// SIMATIC S7-200 SMART project (STEP 7-Micro/WIN SMART), CPU ST40

SYMBOL_TABLE 用户定义1
D1GD             I0.0     // 道1光电
D2GD             I0.1     // 道2光电
D3GD             I0.2     // 道3光电
D4GD             I0.3     // 道4光电
D1YX             I0.4     // 道1运行
D2YX             I0.5     // 道2运行
D3YX             I0.6     // 道3运行
D4YX             I0.7     // 道4运行
END_SYMBOL_TABLE

SYMBOL_TABLE 系统符号
Always_On        SM0.0    // 始终接通
First_Scan_On    SM0.1    // 仅在第一个扫描周期时接通
Clock_1s         SM0.5    // 针对 1 s 的周期时间，时钟脉冲接通 0.5 s，断开 0.5 s.
P0_Config        SMB30    // 组态端口 0 通信：奇偶校验、每个字符的数据位数、波特率和协议
END_SYMBOL_TABLE

SYMBOL_TABLE TCPServer1
State            VB5000
SendBuffer       VB5100
RecvBuffer       VB5300
RecvLenth        VW5004
SendLenth        VW5006
SendBufferW      VW5100
RecvBufferW      VW5300
StateConnect     1
StateConnectWait 2
StateTransmit    3
StateTransmitWait 4
StateReceive     5
StateRecvCheck   6
StateDisconnect  7
StateDisconnectWait 8
ExitSwitch       10
SendLenthB       VB5008
END_SYMBOL_TABLE

ORGANIZATION_BLOCK 主程序:OB1
TITLE=程序注释
BEGIN
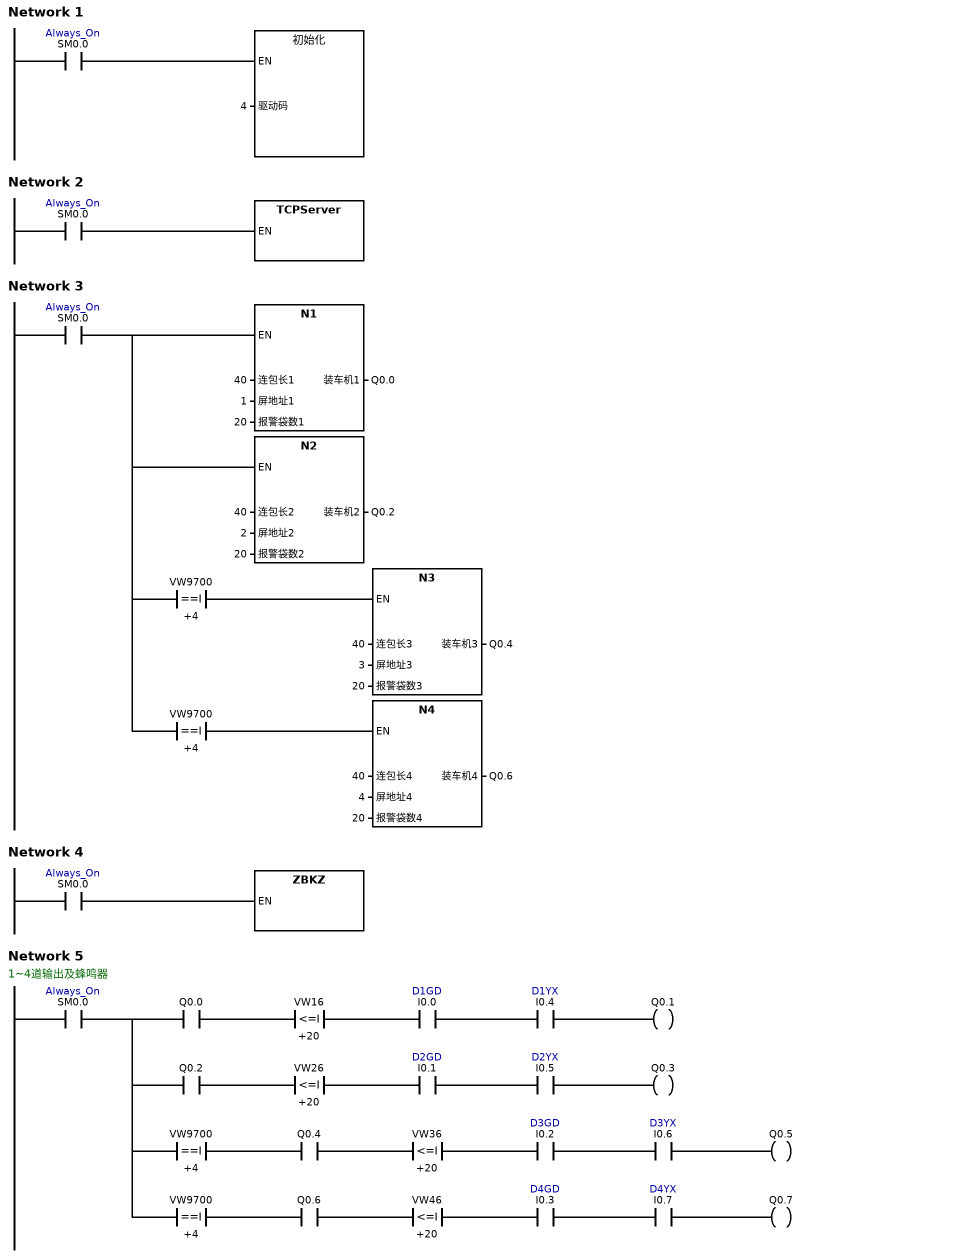
Network 1
LD     Always_On:SM0.0
CALL   初始化:SBR0, 4
Network 2
LD     Always_On:SM0.0
CALL   TCPServer:SBR50
Network 3
LD     Always_On:SM0.0
LPS
CALL   N1:SBR1, 40, 1, 20, Q0.0
CALL   N2:SBR2, 40, 2, 20, Q0.2
AW=    VW9700, +4
CALL   N3:SBR3, 40, 3, 20, Q0.4
LPP
AW=    VW9700, +4
CALL   N4:SBR4, 40, 4, 20, Q0.6
Network 4
LD     Always_On:SM0.0
CALL   ZBKZ:SBR9
Network 5
// 1~4道输出及蜂鸣器
LD     Always_On:SM0.0
LPS
A      Q0.0
AW<=   VW16, +20
A      D1GD:I0.0
A      D1YX:I0.4
=      Q0.1
LRD
A      Q0.2
AW<=   VW26, +20
A      D2GD:I0.1
A      D2YX:I0.5
=      Q0.3
LRD
AW=    VW9700, +4
A      Q0.4
AW<=   VW36, +20
A      D3GD:I0.2
A      D3YX:I0.6
=      Q0.5
LPP
AW=    VW9700, +4
A      Q0.6
AW<=   VW46, +20
A      D4GD:I0.3
A      D4YX:I0.7
=      Q0.7
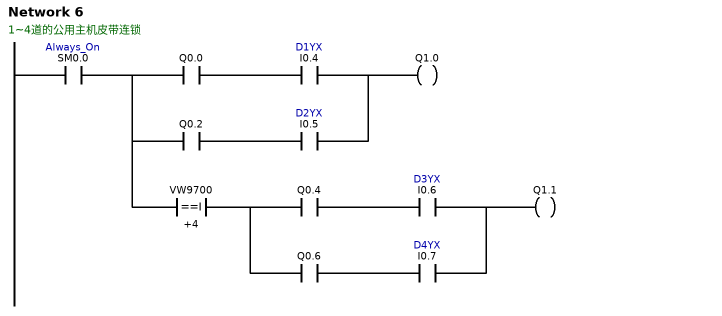
Network 6
// 1~4道的公用主机皮带连锁
LD     Always_On:SM0.0
LPS
LD     Q0.0
A      D1YX:I0.4
LD     Q0.2
A      D2YX:I0.5
OLD
ALD
=      Q1.0
LPP
AW=    VW9700, +4
LD     Q0.4
A      D3YX:I0.6
LD     Q0.6
A      D4YX:I0.7
OLD
ALD
=      Q1.1
END_ORGANIZATION_BLOCK

SUBROUTINE_BLOCK 初始化:SBR0
TITLE=子程序注释
VAR_INPUT
驱动码:WORD;	// LW0 
END_VAR
VAR
temp1:WORD;	// LW2 
temp2:WORD;	// LW4 
END_VAR
BEGIN
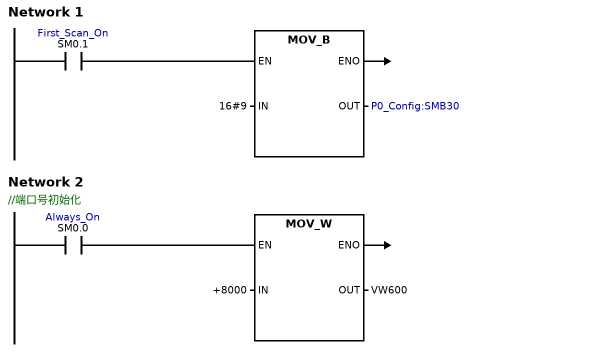
Network 1
// 首次扫描时，
// 初始化自由端口：
// - 选择9600波特
// - 选择8个数据位
// - 选择无校验
// 初始化RCV信息控制字节：
// - RCV被启用
// - 检测到信息字符结束
// - 将空闲行条件检测为
// 信息开始条件。
// 将信息字符结束设为hex OA（换行符）。
// 将空闲行超时设为5毫秒。
// 将最大字符数设为100。
// 为端口0在VB100位置启用带缓冲区的接收方框
LD     First_Scan_On:SM0.1
MOVB   16#9, P0_Config:SMB30
Network 2
// //端口号初始化
LD     Always_On:SM0.0
MOVW   +8000, VW600
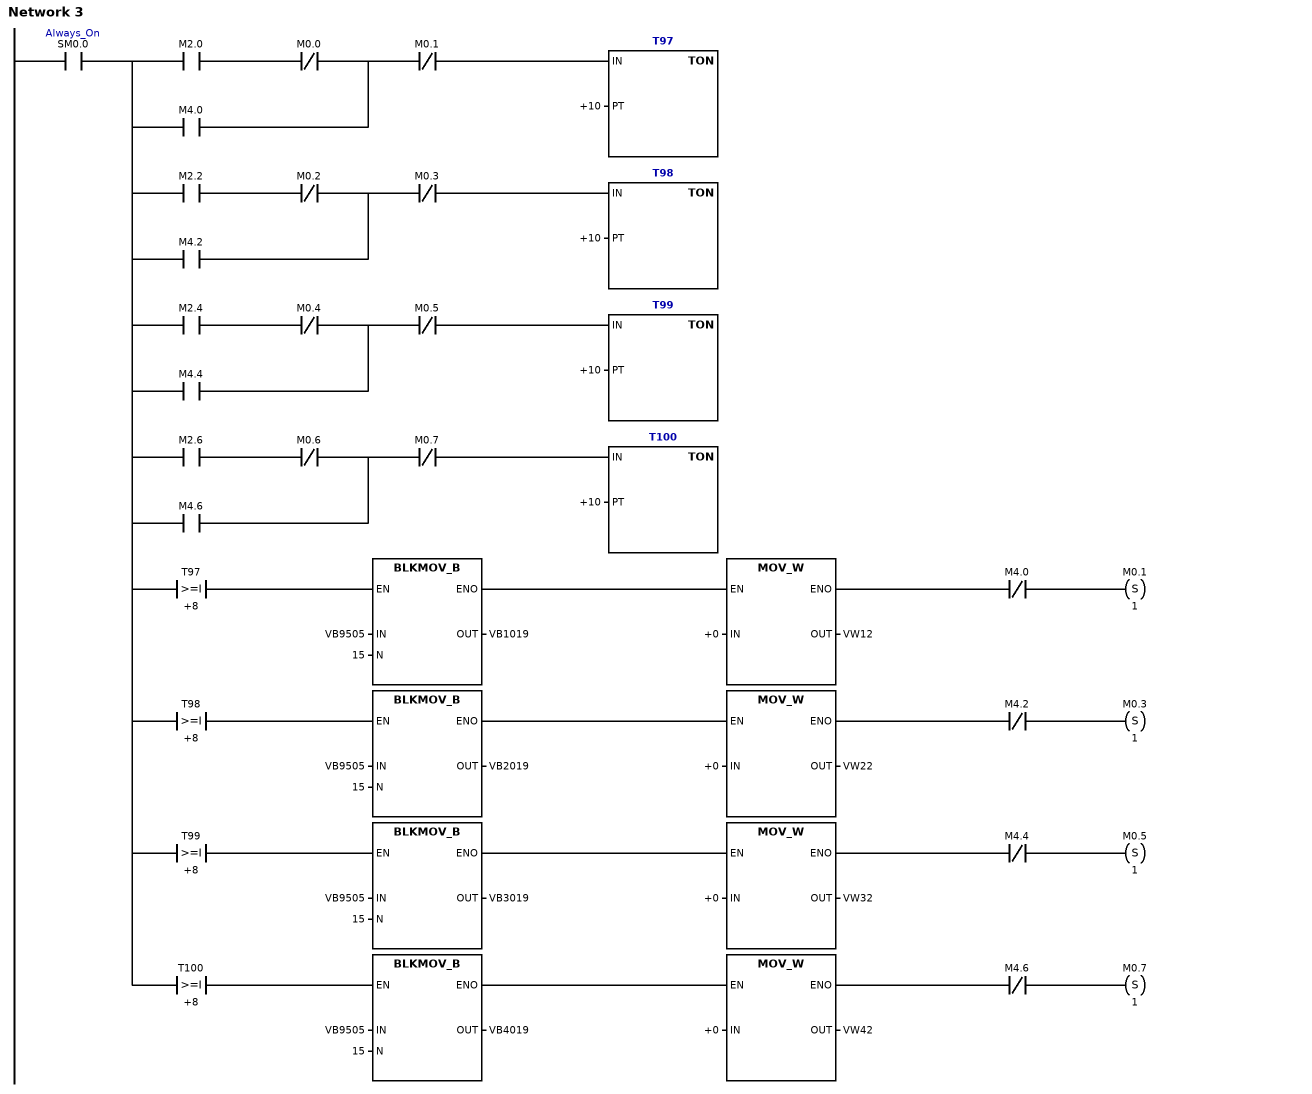
Network 3
LD     Always_On:SM0.0
LPS
LD     M2.0
AN     M0.0
O      M4.0
ALD
AN     M0.1
TON    T97, +10
LRD
LD     M2.2
AN     M0.2
O      M4.2
ALD
AN     M0.3
TON    T98, +10
LRD
LD     M2.4
AN     M0.4
O      M4.4
ALD
AN     M0.5
TON    T99, +10
LRD
LD     M2.6
AN     M0.6
O      M4.6
ALD
AN     M0.7
TON    T100, +10
LPP
LPS
AW>=   T97, +8
BMB    VB9505, VB1019, 15
AENO
MOVW   +0, VW12
AENO
AN     M4.0
S      M0.1, 1
LRD
AW>=   T98, +8
BMB    VB9505, VB2019, 15
AENO
MOVW   +0, VW22
AENO
AN     M4.2
S      M0.3, 1
LRD
AW>=   T99, +8
BMB    VB9505, VB3019, 15
AENO
MOVW   +0, VW32
AENO
AN     M4.4
S      M0.5, 1
LPP
AW>=   T100, +8
BMB    VB9505, VB4019, 15
AENO
MOVW   +0, VW42
AENO
AN     M4.6
S      M0.7, 1
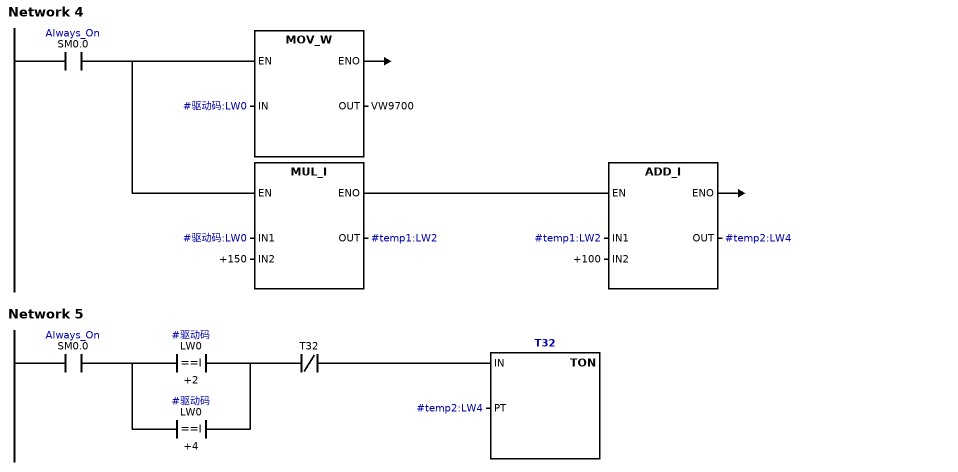
Network 4
LD     Always_On:SM0.0
MOVW   #驱动码:LW0, VW9700
MOVW   #驱动码:LW0, #temp1:LW2
AENO
*I     +150, #temp1:LW2
AENO
MOVW   #temp1:LW2, #temp2:LW4
+I     +100, #temp2:LW4
Network 5
LD     Always_On:SM0.0
LDW=   #驱动码:LW0, +2
OW=    #驱动码:LW0, +4
ALD
AN     T32
TON    T32, #temp2:LW4
END_SUBROUTINE_BLOCK

SUBROUTINE_BLOCK N1:SBR1
TITLE=
VAR_INPUT
连包长1:WORD;	// LW0 
屏地址1:BYTE;	// LB2 
报警袋数1:WORD;	// LW3 
END_VAR
VAR_OUTPUT
装车机1:BOOL;	// L5.0 
END_VAR
VAR
总袋数1:WORD;	// LW6 
袋长1:WORD;	// LW8 
已装袋数1:WORD;	// LW10 
剩余袋数1:WORD;	// LW12 
END_VAR
BEGIN
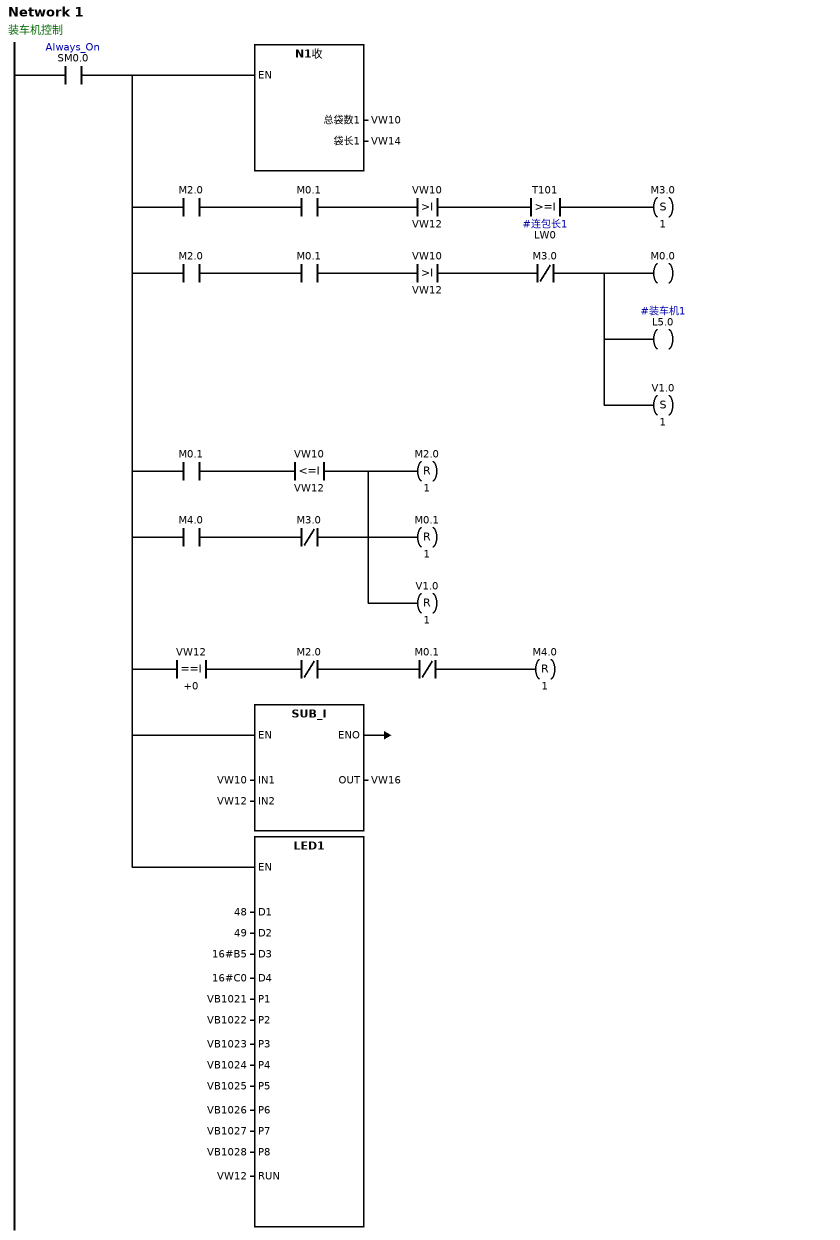
Network 1
// 装车机控制
LD     Always_On:SM0.0
LPS
CALL   N1收:SBR21, VW10, VW14
A      M2.0
A      M0.1
AW>    VW10, VW12
AW>=   T101, #连包长1:LW0
S      M3.0, 1
LRD
A      M2.0
A      M0.1
AW>    VW10, VW12
AN     M3.0
=      M0.0
=      #装车机1:L5.0
S      V1.0, 1
LRD
LD     M0.1
AW<=   VW10, VW12
LD     M4.0
AN     M3.0
OLD
ALD
R      M2.0, 1
R      M0.1, 1
R      V1.0, 1
LPP
LPS
AW=    VW12, +0
AN     M2.0
AN     M0.1
R      M4.0, 1
LRD
MOVW   VW10, VW16
-I     VW12, VW16
LPP
CALL   LED1:SBR11, 48, 49, 16#B5, 16#C0, VB1021, VB1022, VB1023, VB1024, VB1025, VB1026, VB1027, VB1028, VW12
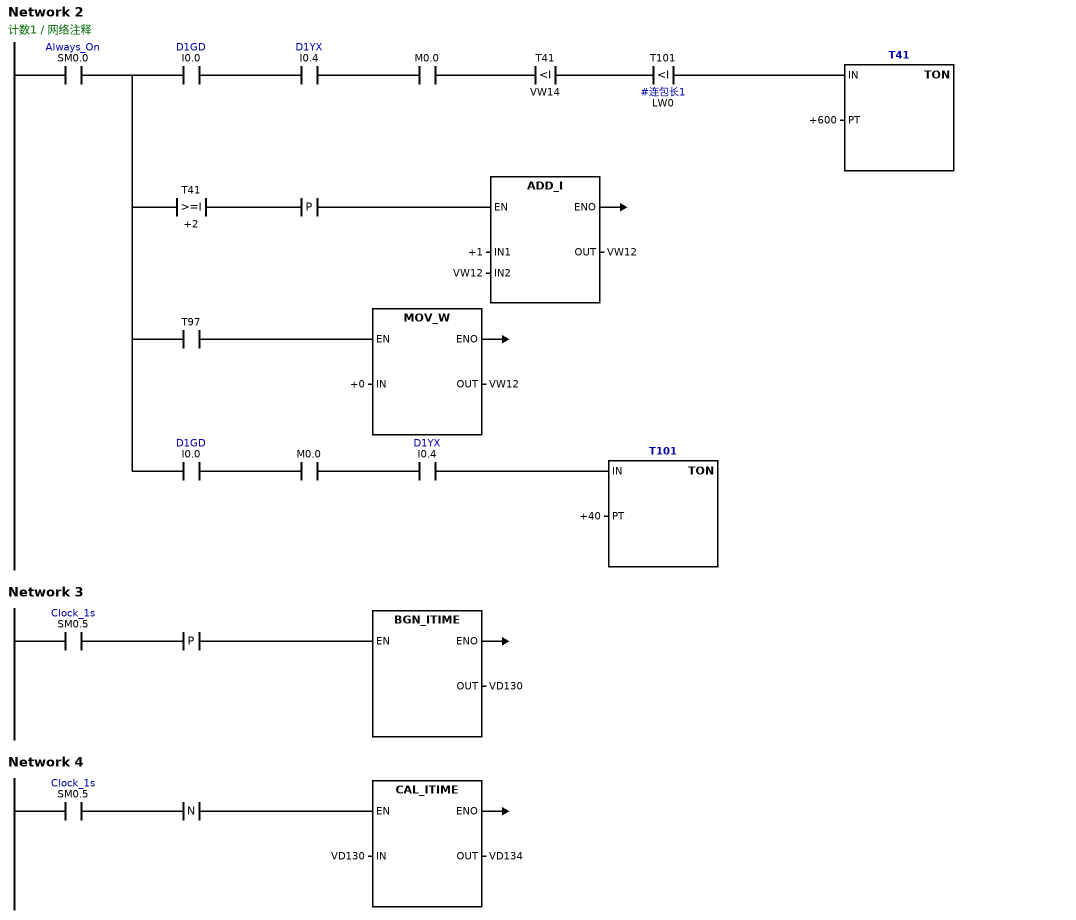
Network 2
// 计数1
// 网络注释
LD     Always_On:SM0.0
LPS
A      D1GD:I0.0
A      D1YX:I0.4
A      M0.0
AW<    T41, VW14
AW<    T101, #连包长1:LW0
TON    T41, +600
LRD
AW>=   T41, +2
EU
+I     +1, VW12
LRD
A      T97
MOVW   +0, VW12
LPP
A      D1GD:I0.0
A      M0.0
A      D1YX:I0.4
TON    T101, +40
Network 3
LD     Clock_1s:SM0.5
EU
BITIM  VD130
Network 4
LD     Clock_1s:SM0.5
ED
CITIM  VD130, VD134
END_SUBROUTINE_BLOCK

SUBROUTINE_BLOCK N2:SBR2
TITLE=
VAR_INPUT
连包长2:WORD;	// LW0 
屏地址2:BYTE;	// LB2 
报警袋数2:WORD;	// LW3 
END_VAR
VAR_OUTPUT
装车机2:BOOL;	// L5.0 
END_VAR
VAR
总袋数2:WORD;	// LW6 
袋长2:WORD;	// LW8 
已装袋数2:WORD;	// LW10 
剩余袋数2:WORD;	// LW12 
END_VAR
BEGIN
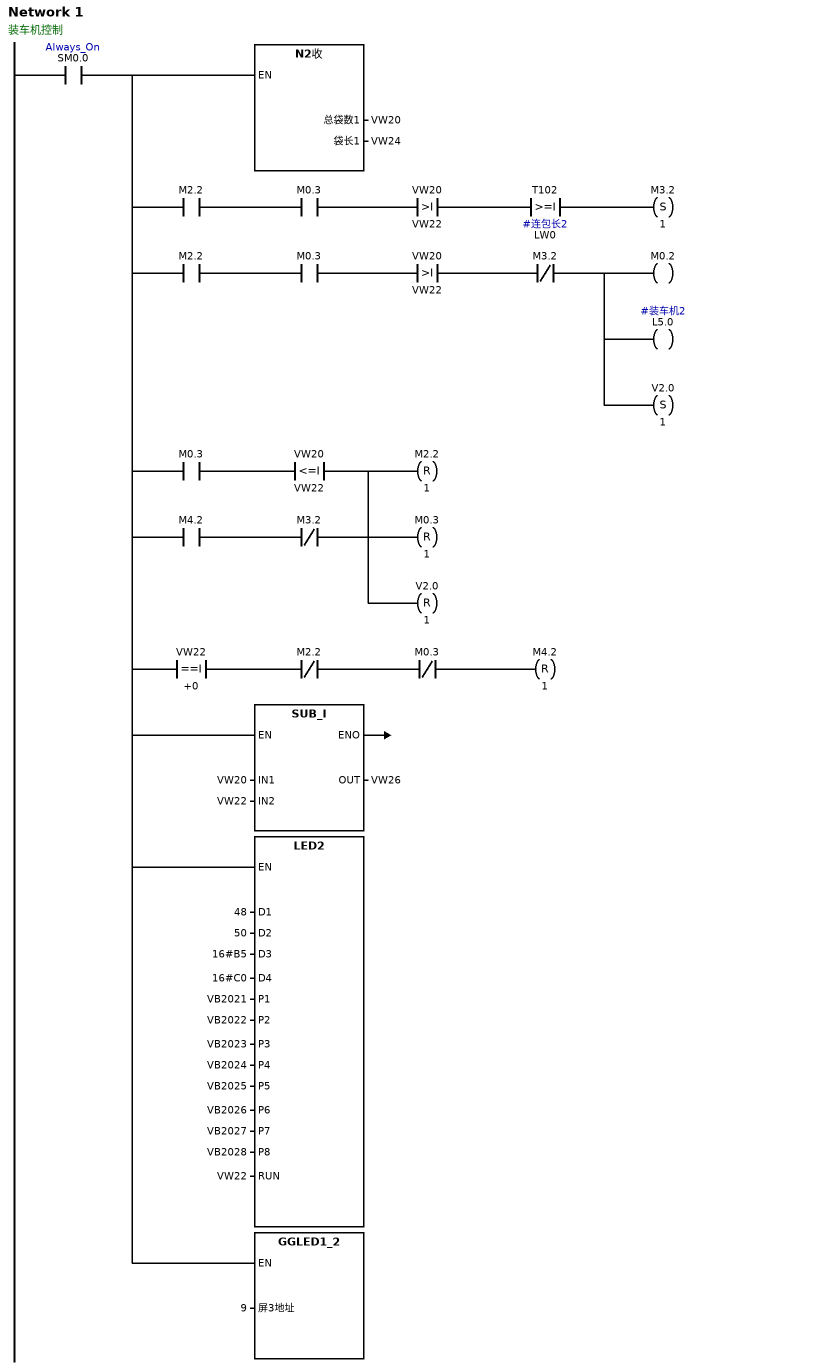
Network 1
// 装车机控制
LD     Always_On:SM0.0
LPS
CALL   N2收:SBR22, VW20, VW24
A      M2.2
A      M0.3
AW>    VW20, VW22
AW>=   T102, #连包长2:LW0
S      M3.2, 1
LRD
A      M2.2
A      M0.3
AW>    VW20, VW22
AN     M3.2
=      M0.2
=      #装车机2:L5.0
S      V2.0, 1
LRD
LD     M0.3
AW<=   VW20, VW22
LD     M4.2
AN     M3.2
OLD
ALD
R      M2.2, 1
R      M0.3, 1
R      V2.0, 1
LPP
LPS
AW=    VW22, +0
AN     M2.2
AN     M0.3
R      M4.2, 1
LRD
MOVW   VW20, VW26
-I     VW22, VW26
LRD
CALL   LED2:SBR12, 48, 50, 16#B5, 16#C0, VB2021, VB2022, VB2023, VB2024, VB2025, VB2026, VB2027, VB2028, VW22
LPP
CALL   GGLED1_2:SBR31, 9
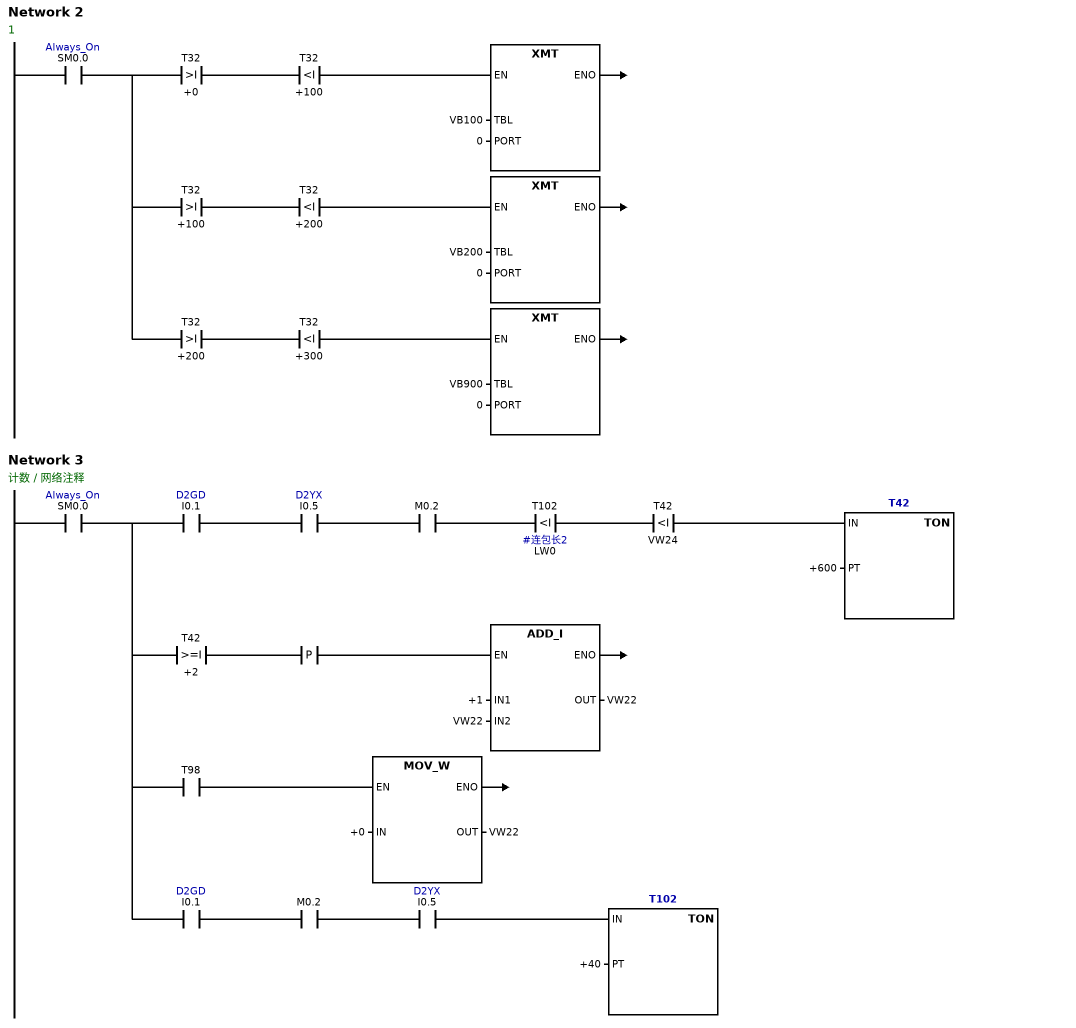
Network 2
// 1
LD     Always_On:SM0.0
LPS
AW>    T32, +0
AW<    T32, +100
XMT    VB100, 0
LRD
AW>    T32, +100
AW<    T32, +200
XMT    VB200, 0
LPP
AW>    T32, +200
AW<    T32, +300
XMT    VB900, 0
Network 3
// 计数
// 网络注释
LD     Always_On:SM0.0
LPS
A      D2GD:I0.1
A      D2YX:I0.5
A      M0.2
AW<    T102, #连包长2:LW0
AW<    T42, VW24
TON    T42, +600
LRD
AW>=   T42, +2
EU
+I     +1, VW22
LRD
A      T98
MOVW   +0, VW22
LPP
A      D2GD:I0.1
A      M0.2
A      D2YX:I0.5
TON    T102, +40
END_SUBROUTINE_BLOCK

SUBROUTINE_BLOCK N3:SBR3
TITLE=
VAR_INPUT
连包长3:WORD;	// LW0 
屏地址3:BYTE;	// LB2 
报警袋数3:WORD;	// LW3 
END_VAR
VAR_OUTPUT
装车机3:BOOL;	// L5.0 
END_VAR
VAR
总袋数3:WORD;	// LW6 
袋长3:WORD;	// LW8 
已装袋数3:WORD;	// LW10 
剩余袋数3:WORD;	// LW12 
END_VAR
BEGIN
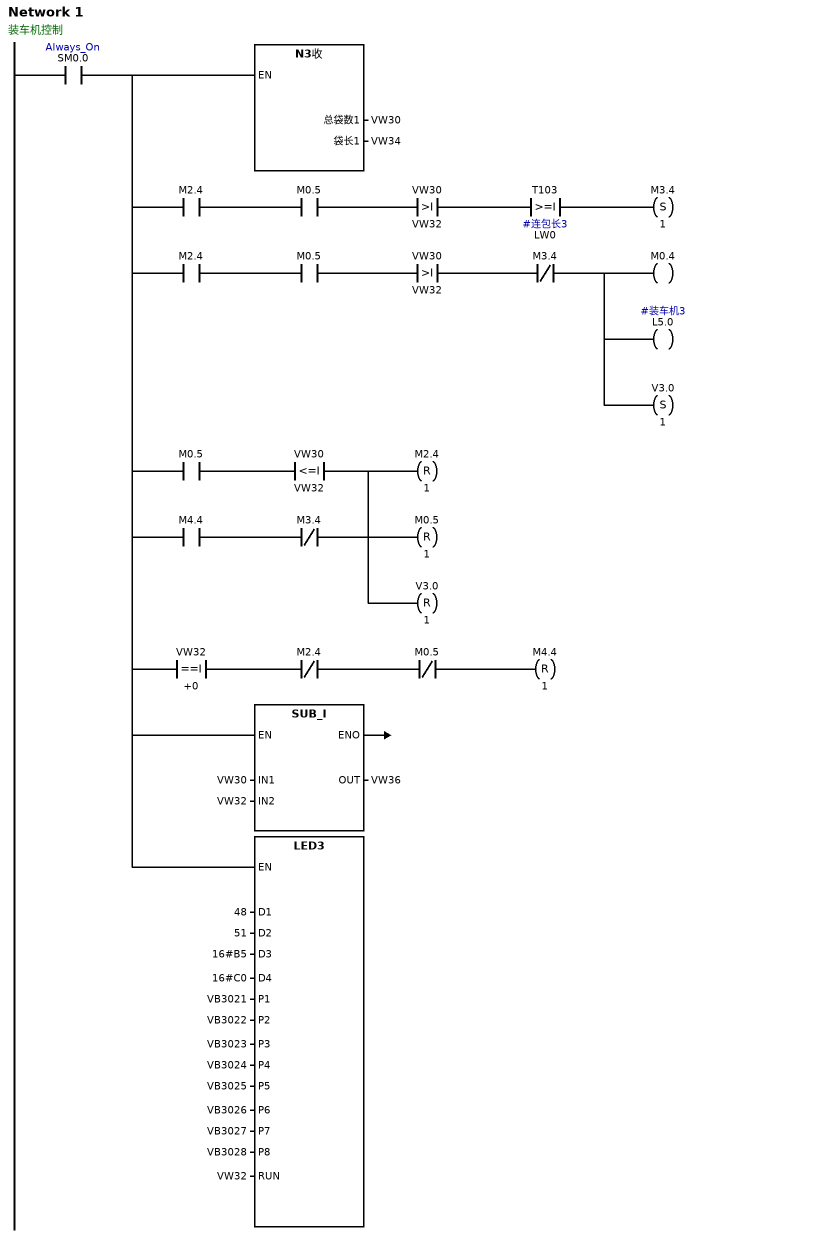
Network 1
// 装车机控制
LD     Always_On:SM0.0
LPS
CALL   N3收:SBR23, VW30, VW34
A      M2.4
A      M0.5
AW>    VW30, VW32
AW>=   T103, #连包长3:LW0
S      M3.4, 1
LRD
A      M2.4
A      M0.5
AW>    VW30, VW32
AN     M3.4
=      M0.4
=      #装车机3:L5.0
S      V3.0, 1
LRD
LD     M0.5
AW<=   VW30, VW32
LD     M4.4
AN     M3.4
OLD
ALD
R      M2.4, 1
R      M0.5, 1
R      V3.0, 1
LPP
LPS
AW=    VW32, +0
AN     M2.4
AN     M0.5
R      M4.4, 1
LRD
MOVW   VW30, VW36
-I     VW32, VW36
LPP
CALL   LED3:SBR13, 48, 51, 16#B5, 16#C0, VB3021, VB3022, VB3023, VB3024, VB3025, VB3026, VB3027, VB3028, VW32
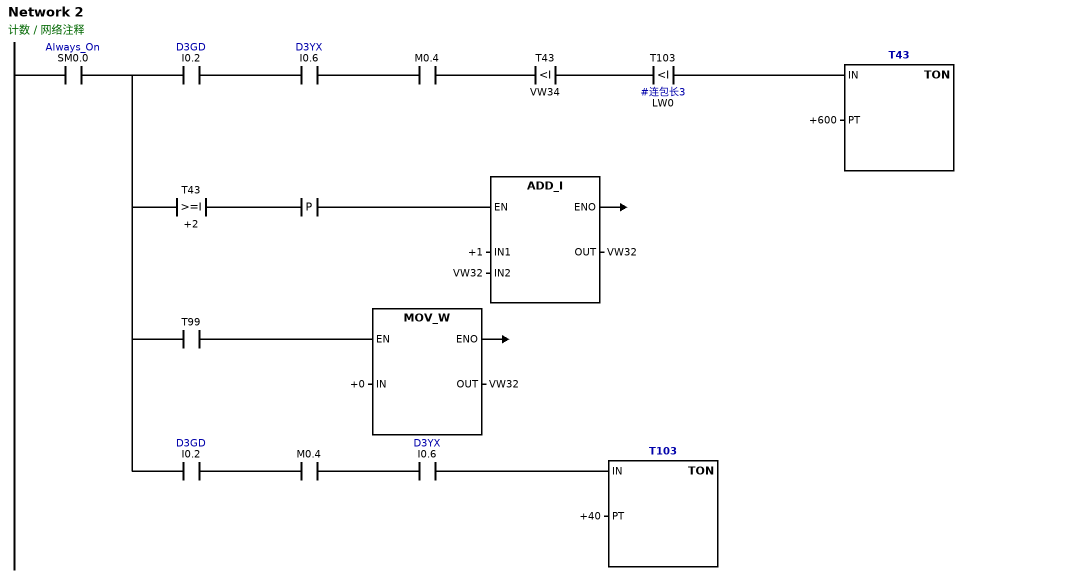
Network 2
// 计数
// 网络注释
LD     Always_On:SM0.0
LPS
A      D3GD:I0.2
A      D3YX:I0.6
A      M0.4
AW<    T43, VW34
AW<    T103, #连包长3:LW0
TON    T43, +600
LRD
AW>=   T43, +2
EU
+I     +1, VW32
LRD
A      T99
MOVW   +0, VW32
LPP
A      D3GD:I0.2
A      M0.4
A      D3YX:I0.6
TON    T103, +40
END_SUBROUTINE_BLOCK

SUBROUTINE_BLOCK N4:SBR4
TITLE=
VAR_INPUT
连包长4:WORD;	// LW0 
屏地址4:BYTE;	// LB2 
报警袋数4:WORD;	// LW3 
END_VAR
VAR_OUTPUT
装车机4:BOOL;	// L5.0 
END_VAR
VAR
总袋数4:WORD;	// LW6 
袋长4:WORD;	// LW8 
已装袋数4:WORD;	// LW10 
剩余袋数4:WORD;	// LW12 
END_VAR
BEGIN
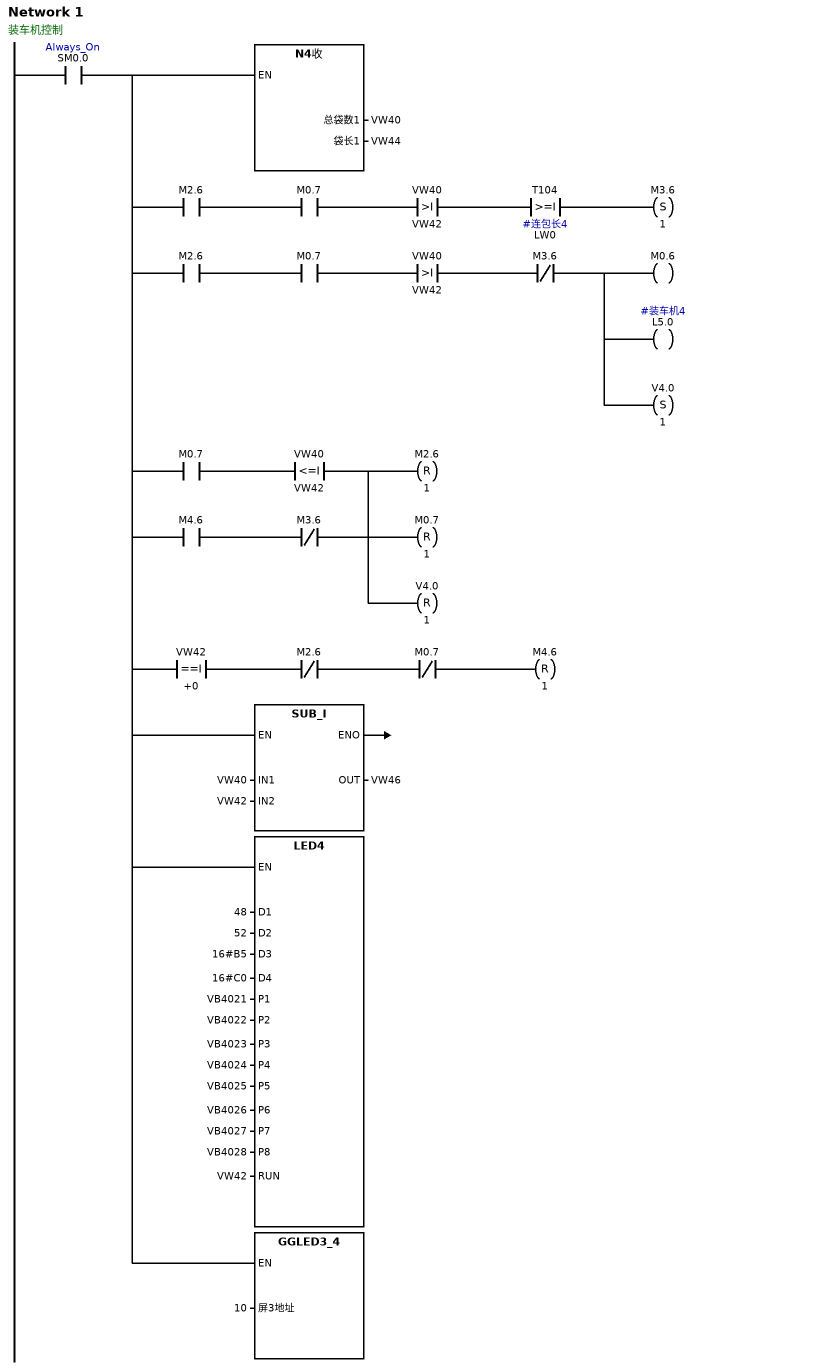
Network 1
// 装车机控制
LD     Always_On:SM0.0
LPS
CALL   N4收:SBR24, VW40, VW44
A      M2.6
A      M0.7
AW>    VW40, VW42
AW>=   T104, #连包长4:LW0
S      M3.6, 1
LRD
A      M2.6
A      M0.7
AW>    VW40, VW42
AN     M3.6
=      M0.6
=      #装车机4:L5.0
S      V4.0, 1
LRD
LD     M0.7
AW<=   VW40, VW42
LD     M4.6
AN     M3.6
OLD
ALD
R      M2.6, 1
R      M0.7, 1
R      V4.0, 1
LPP
LPS
AW=    VW42, +0
AN     M2.6
AN     M0.7
R      M4.6, 1
LRD
MOVW   VW40, VW46
-I     VW42, VW46
LRD
CALL   LED4:SBR14, 48, 52, 16#B5, 16#C0, VB4021, VB4022, VB4023, VB4024, VB4025, VB4026, VB4027, VB4028, VW42
LPP
CALL   GGLED3_4:SBR32, 10
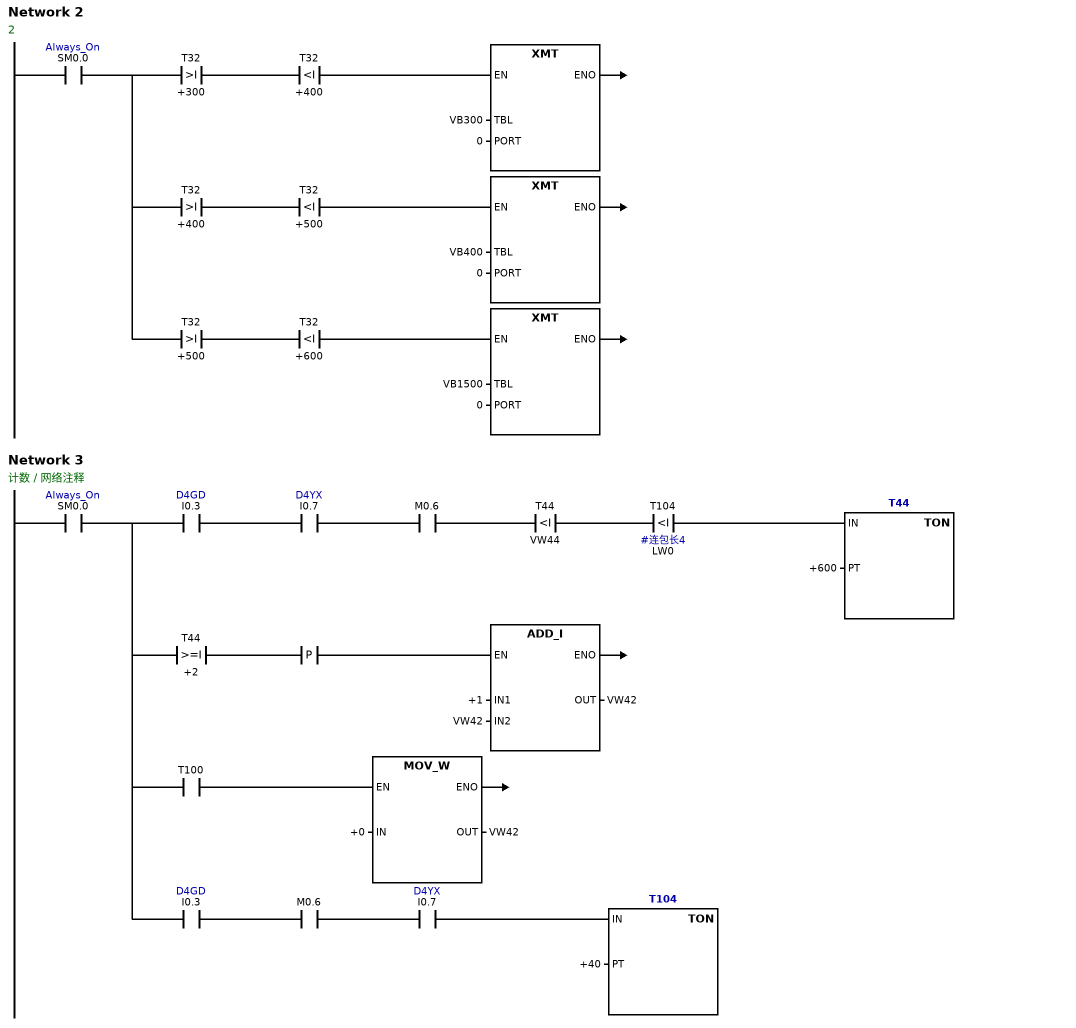
Network 2
// 2
LD     Always_On:SM0.0
LPS
AW>    T32, +300
AW<    T32, +400
XMT    VB300, 0
LRD
AW>    T32, +400
AW<    T32, +500
XMT    VB400, 0
LPP
AW>    T32, +500
AW<    T32, +600
XMT    VB1500, 0
Network 3
// 计数
// 网络注释
LD     Always_On:SM0.0
LPS
A      D4GD:I0.3
A      D4YX:I0.7
A      M0.6
AW<    T44, VW44
AW<    T104, #连包长4:LW0
TON    T44, +600
LRD
AW>=   T44, +2
EU
+I     +1, VW42
LRD
A      T100
MOVW   +0, VW42
LPP
A      D4GD:I0.3
A      M0.6
A      D4YX:I0.7
TON    T104, +40
END_SUBROUTINE_BLOCK

// SBR5: protected block, not included

// SBR6: protected block, not included

// SBR7: protected block, not included

// SBR8: protected block, not included

SUBROUTINE_BLOCK ZBKZ:SBR9
TITLE=子程序注释
BEGIN
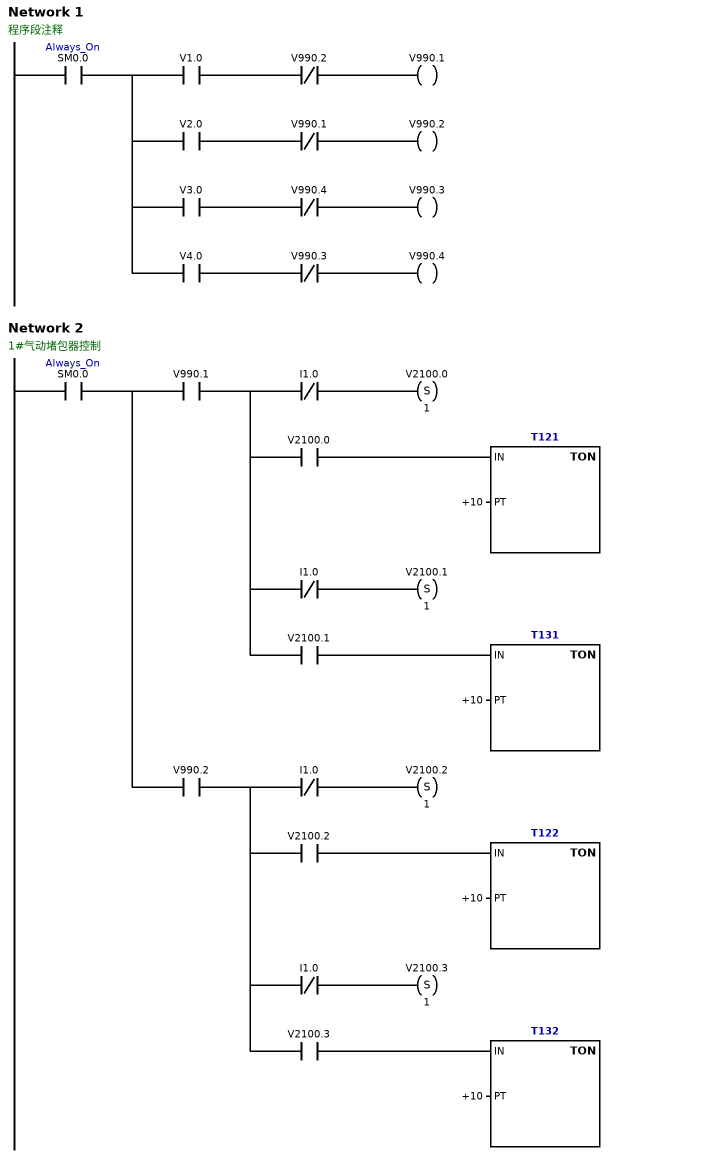
Network 1
// 程序段注释
LD     Always_On:SM0.0
LPS
A      V1.0
AN     V990.2
=      V990.1
LRD
A      V2.0
AN     V990.1
=      V990.2
LRD
A      V3.0
AN     V990.4
=      V990.3
LPP
A      V4.0
AN     V990.3
=      V990.4
Network 2
// 1#气动堵包器控制
LD     Always_On:SM0.0
LPS
A      V990.1
LPS
AN     I1.0
S      V2100.0, 1
LRD
A      V2100.0
TON    T121, +10
LRD
AN     I1.0
S      V2100.1, 1
LPP
A      V2100.1
TON    T131, +10
LPP
A      V990.2
LPS
AN     I1.0
S      V2100.2, 1
LRD
A      V2100.2
TON    T122, +10
LRD
AN     I1.0
S      V2100.3, 1
LPP
A      V2100.3
TON    T132, +10
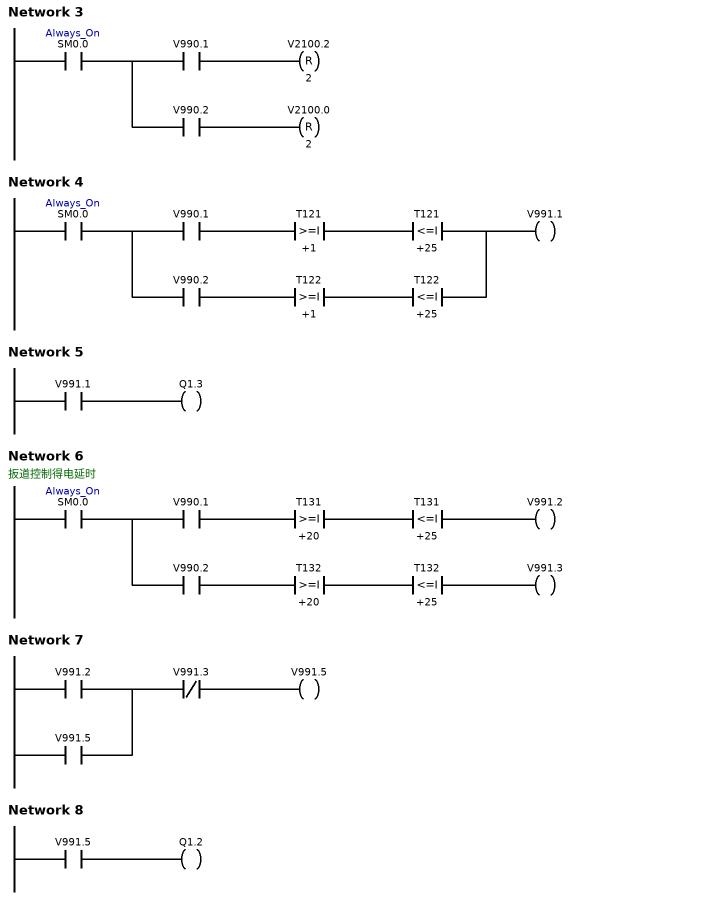
Network 3
LD     Always_On:SM0.0
LPS
A      V990.1
R      V2100.2, 2
LPP
A      V990.2
R      V2100.0, 2
Network 4
LD     Always_On:SM0.0
LD     V990.1
AW>=   T121, +1
AW<=   T121, +25
LD     V990.2
AW>=   T122, +1
AW<=   T122, +25
OLD
ALD
=      V991.1
Network 5
LD     V991.1
=      Q1.3
Network 6
// 扳道控制得电延时
LD     Always_On:SM0.0
LPS
A      V990.1
AW>=   T131, +20
AW<=   T131, +25
=      V991.2
LPP
A      V990.2
AW>=   T132, +20
AW<=   T132, +25
=      V991.3
Network 7
LD     V991.2
O      V991.5
AN     V991.3
=      V991.5
Network 8
LD     V991.5
=      Q1.2
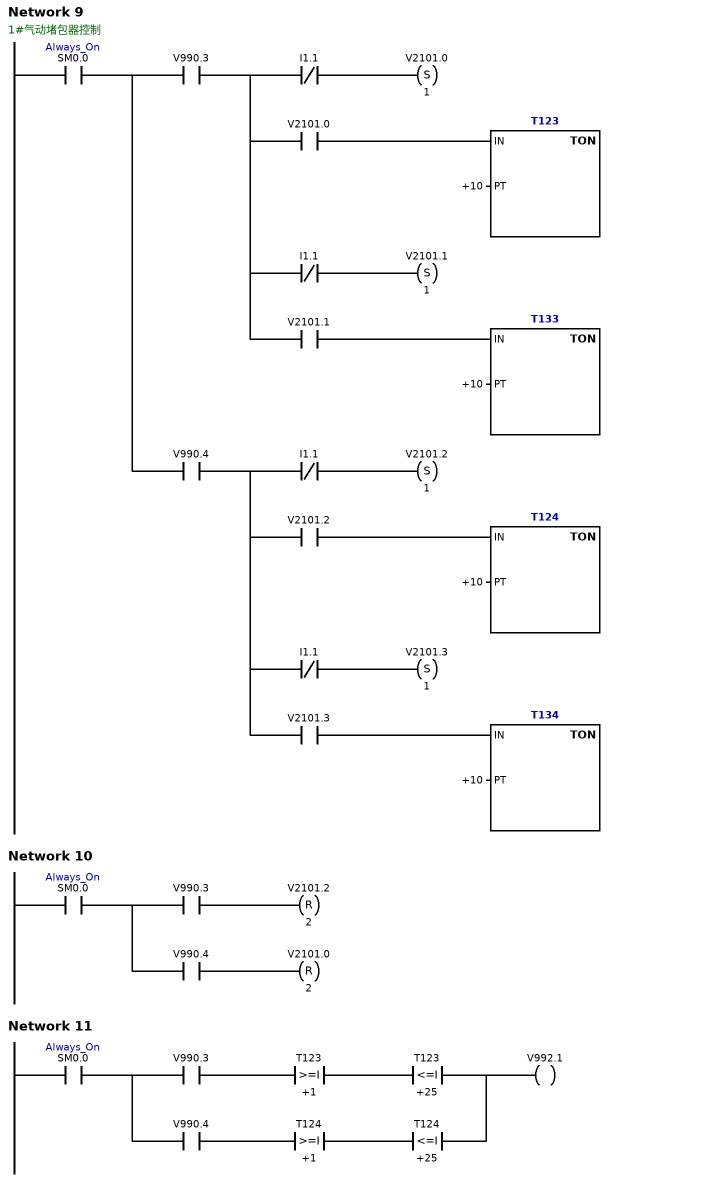
Network 9
// 1#气动堵包器控制
LD     Always_On:SM0.0
LPS
A      V990.3
LPS
AN     I1.1
S      V2101.0, 1
LRD
A      V2101.0
TON    T123, +10
LRD
AN     I1.1
S      V2101.1, 1
LPP
A      V2101.1
TON    T133, +10
LPP
A      V990.4
LPS
AN     I1.1
S      V2101.2, 1
LRD
A      V2101.2
TON    T124, +10
LRD
AN     I1.1
S      V2101.3, 1
LPP
A      V2101.3
TON    T134, +10
Network 10
LD     Always_On:SM0.0
LPS
A      V990.3
R      V2101.2, 2
LPP
A      V990.4
R      V2101.0, 2
Network 11
LD     Always_On:SM0.0
LD     V990.3
AW>=   T123, +1
AW<=   T123, +25
LD     V990.4
AW>=   T124, +1
AW<=   T124, +25
OLD
ALD
=      V992.1
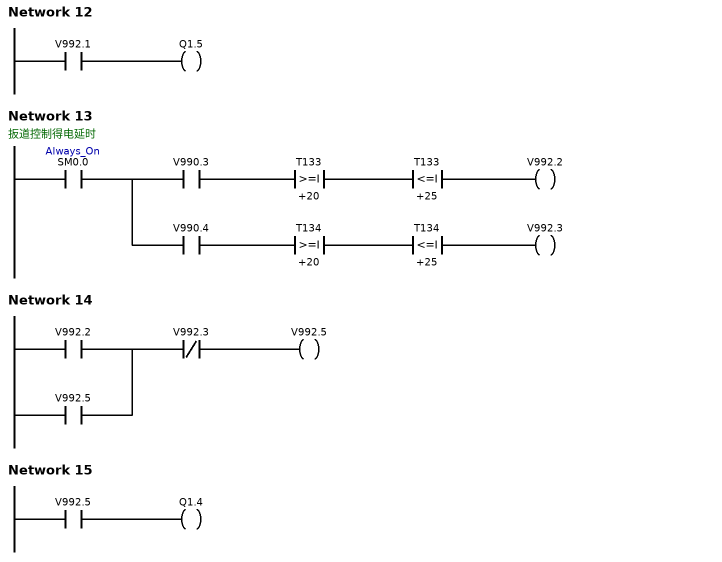
Network 12
LD     V992.1
=      Q1.5
Network 13
// 扳道控制得电延时
LD     Always_On:SM0.0
LPS
A      V990.3
AW>=   T133, +20
AW<=   T133, +25
=      V992.2
LPP
A      V990.4
AW>=   T134, +20
AW<=   T134, +25
=      V992.3
Network 14
LD     V992.2
O      V992.5
AN     V992.3
=      V992.5
Network 15
LD     V992.5
=      Q1.4
END_SUBROUTINE_BLOCK

SUBROUTINE_BLOCK LED1:SBR11
TITLE=
VAR_INPUT
D1:BYTE;	// LB0 
D2:BYTE;	// LB1 
D3:BYTE;	// LB2 
D4:BYTE;	// LB3 
P1:BYTE;	// LB4 
P2:BYTE;	// LB5 
P3:BYTE;	// LB6 
P4:BYTE;	// LB7 
P5:BYTE;	// LB8 
P6:BYTE;	// LB9 
P7:BYTE;	// LB10 
P8:BYTE;	// LB11 
RUN:WORD;	// LW12 
END_VAR
BEGIN
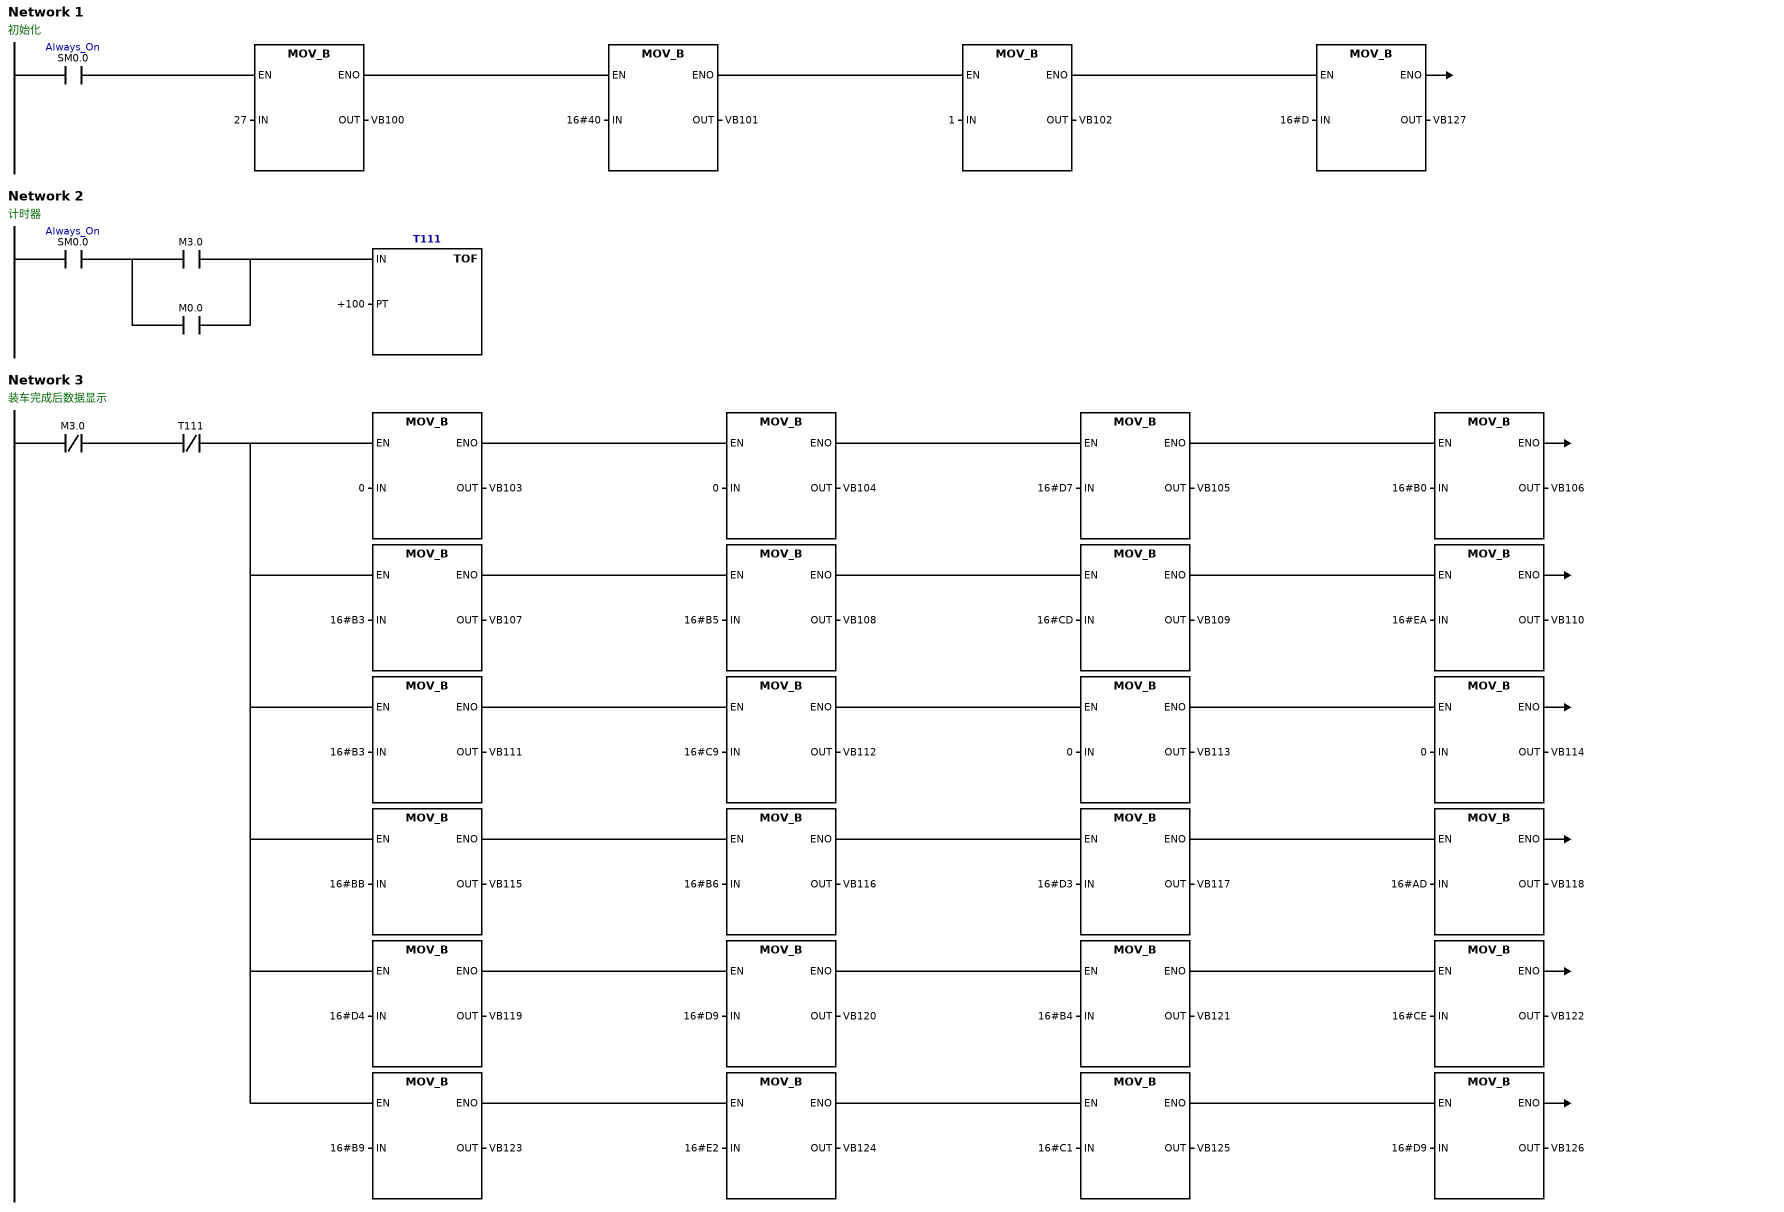
Network 1
// 初始化
LD     Always_On:SM0.0
MOVB   27, VB100
AENO
MOVB   16#40, VB101
AENO
MOVB   1, VB102
AENO
MOVB   16#D, VB127
Network 2
// 计时器
LD     Always_On:SM0.0
LD     M3.0
O      M0.0
ALD
TOF    T111, +100
Network 3
// 装车完成后数据显示
LDN    M3.0
AN     T111
LPS
MOVB   0, VB103
AENO
MOVB   0, VB104
AENO
MOVB   16#D7, VB105
AENO
MOVB   16#B0, VB106
LRD
MOVB   16#B3, VB107
AENO
MOVB   16#B5, VB108
AENO
MOVB   16#CD, VB109
AENO
MOVB   16#EA, VB110
LRD
MOVB   16#B3, VB111
AENO
MOVB   16#C9, VB112
AENO
MOVB   0, VB113
AENO
MOVB   0, VB114
LRD
MOVB   16#BB, VB115
AENO
MOVB   16#B6, VB116
AENO
MOVB   16#D3, VB117
AENO
MOVB   16#AD, VB118
LRD
MOVB   16#D4, VB119
AENO
MOVB   16#D9, VB120
AENO
MOVB   16#B4, VB121
AENO
MOVB   16#CE, VB122
LPP
MOVB   16#B9, VB123
AENO
MOVB   16#E2, VB124
AENO
MOVB   16#C1, VB125
AENO
MOVB   16#D9, VB126
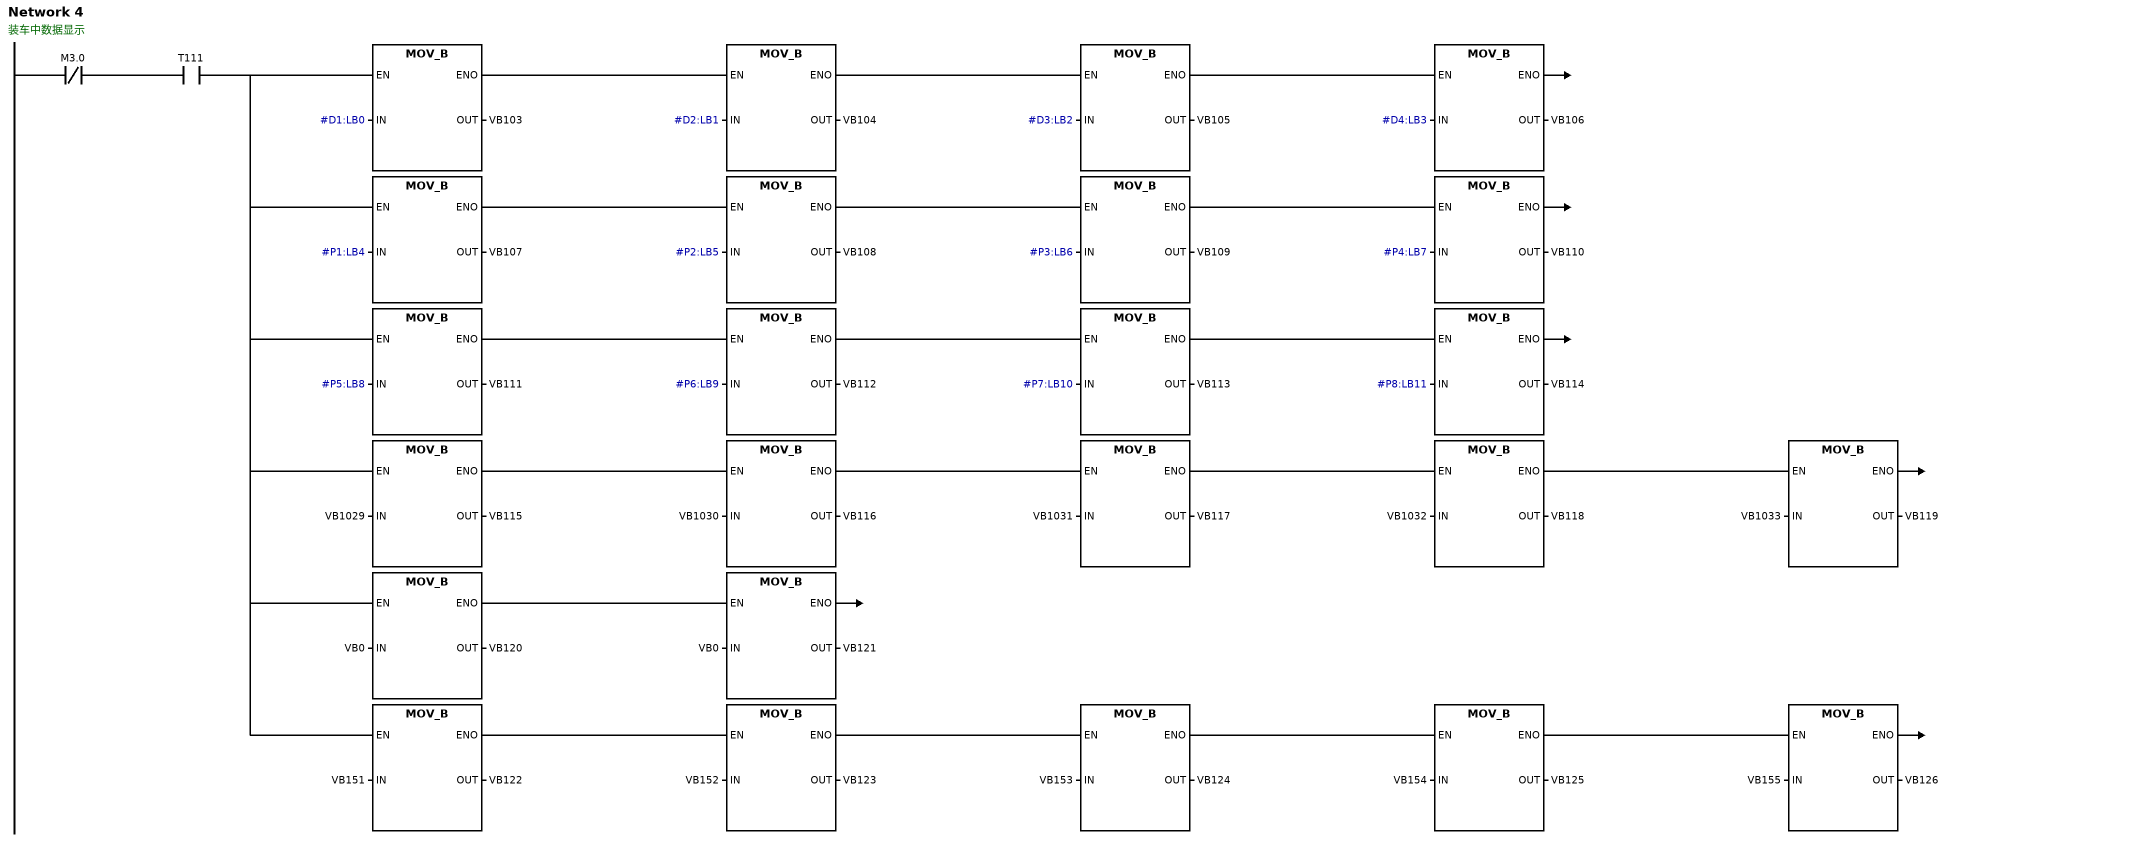
Network 4
// 装车中数据显示
LDN    M3.0
A      T111
LPS
MOVB   #D1:LB0, VB103
AENO
MOVB   #D2:LB1, VB104
AENO
MOVB   #D3:LB2, VB105
AENO
MOVB   #D4:LB3, VB106
LRD
MOVB   #P1:LB4, VB107
AENO
MOVB   #P2:LB5, VB108
AENO
MOVB   #P3:LB6, VB109
AENO
MOVB   #P4:LB7, VB110
LRD
MOVB   #P5:LB8, VB111
AENO
MOVB   #P6:LB9, VB112
AENO
MOVB   #P7:LB10, VB113
AENO
MOVB   #P8:LB11, VB114
LRD
MOVB   VB1029, VB115
AENO
MOVB   VB1030, VB116
AENO
MOVB   VB1031, VB117
AENO
MOVB   VB1032, VB118
AENO
MOVB   VB1033, VB119
LRD
MOVB   VB0, VB120
AENO
MOVB   VB0, VB121
LPP
MOVB   VB151, VB122
AENO
MOVB   VB152, VB123
AENO
MOVB   VB153, VB124
AENO
MOVB   VB154, VB125
AENO
MOVB   VB155, VB126
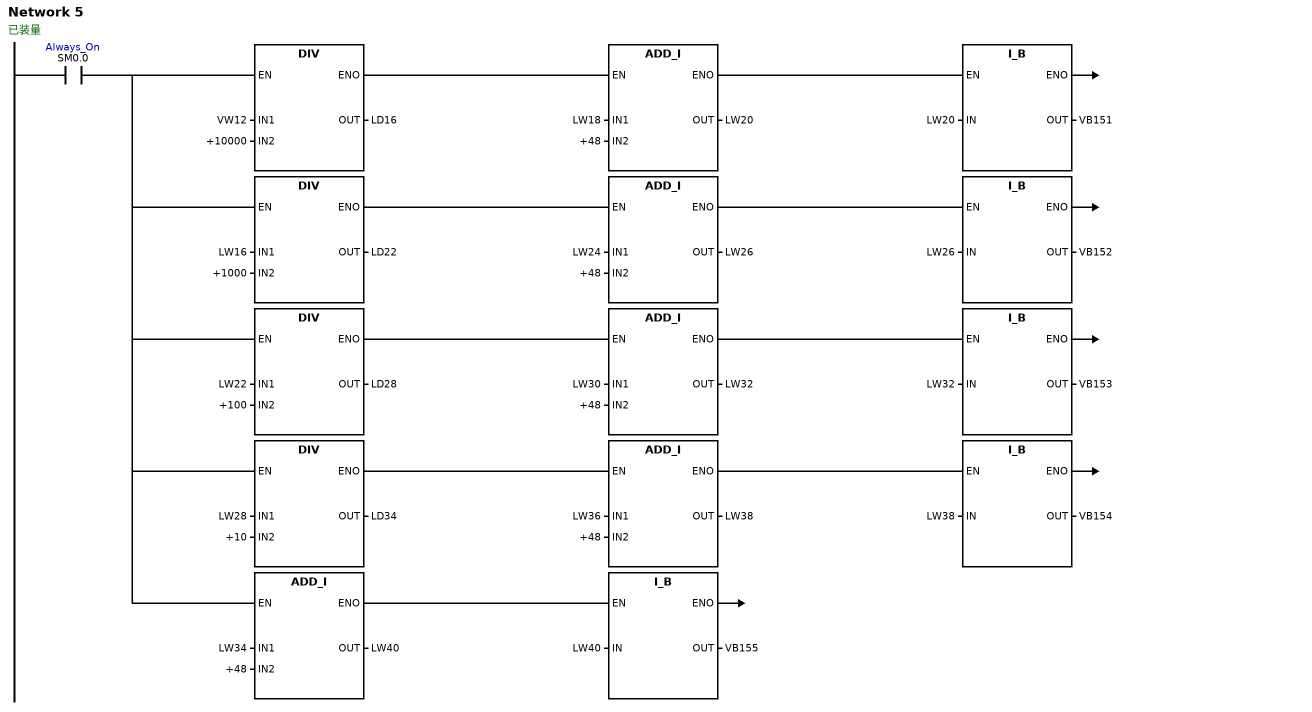
Network 5
// 已装量
LD     Always_On:SM0.0
LPS
MOVW   VW12, LW18
AENO
DIV    +10000, LD16
AENO
MOVW   LW18, LW20
AENO
+I     +48, LW20
AENO
ITB    LW20, VB151
LRD
MOVW   LW16, LW24
AENO
DIV    +1000, LD22
AENO
MOVW   LW24, LW26
AENO
+I     +48, LW26
AENO
ITB    LW26, VB152
LRD
MOVW   LW22, LW30
AENO
DIV    +100, LD28
AENO
MOVW   LW30, LW32
AENO
+I     +48, LW32
AENO
ITB    LW32, VB153
LRD
MOVW   LW28, LW36
AENO
DIV    +10, LD34
AENO
MOVW   LW36, LW38
AENO
+I     +48, LW38
AENO
ITB    LW38, VB154
LPP
MOVW   LW34, LW40
AENO
+I     +48, LW40
AENO
ITB    LW40, VB155
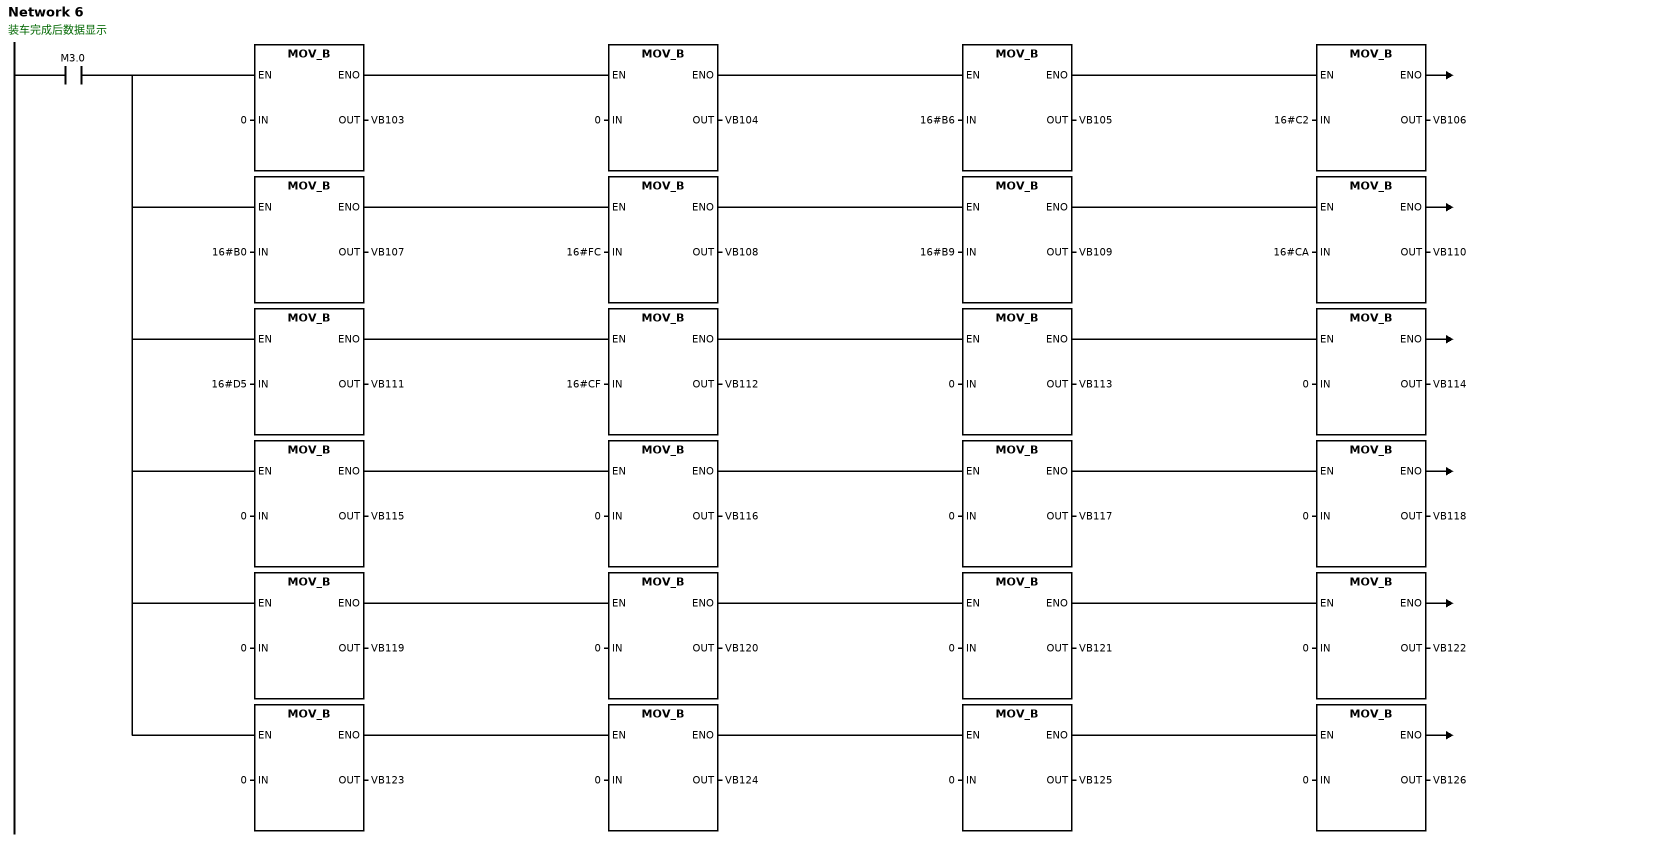
Network 6
// 装车完成后数据显示
LD     M3.0
LPS
MOVB   0, VB103
AENO
MOVB   0, VB104
AENO
MOVB   16#B6, VB105
AENO
MOVB   16#C2, VB106
LRD
MOVB   16#B0, VB107
AENO
MOVB   16#FC, VB108
AENO
MOVB   16#B9, VB109
AENO
MOVB   16#CA, VB110
LRD
MOVB   16#D5, VB111
AENO
MOVB   16#CF, VB112
AENO
MOVB   0, VB113
AENO
MOVB   0, VB114
LRD
MOVB   0, VB115
AENO
MOVB   0, VB116
AENO
MOVB   0, VB117
AENO
MOVB   0, VB118
LRD
MOVB   0, VB119
AENO
MOVB   0, VB120
AENO
MOVB   0, VB121
AENO
MOVB   0, VB122
LPP
MOVB   0, VB123
AENO
MOVB   0, VB124
AENO
MOVB   0, VB125
AENO
MOVB   0, VB126
END_SUBROUTINE_BLOCK

SUBROUTINE_BLOCK LED2:SBR12
TITLE=
VAR_INPUT
D1:BYTE;	// LB0 
D2:BYTE;	// LB1 
D3:BYTE;	// LB2 
D4:BYTE;	// LB3 
P1:BYTE;	// LB4 
P2:BYTE;	// LB5 
P3:BYTE;	// LB6 
P4:BYTE;	// LB7 
P5:BYTE;	// LB8 
P6:BYTE;	// LB9 
P7:BYTE;	// LB10 
P8:BYTE;	// LB11 
RUN:WORD;	// LW12 
END_VAR
BEGIN
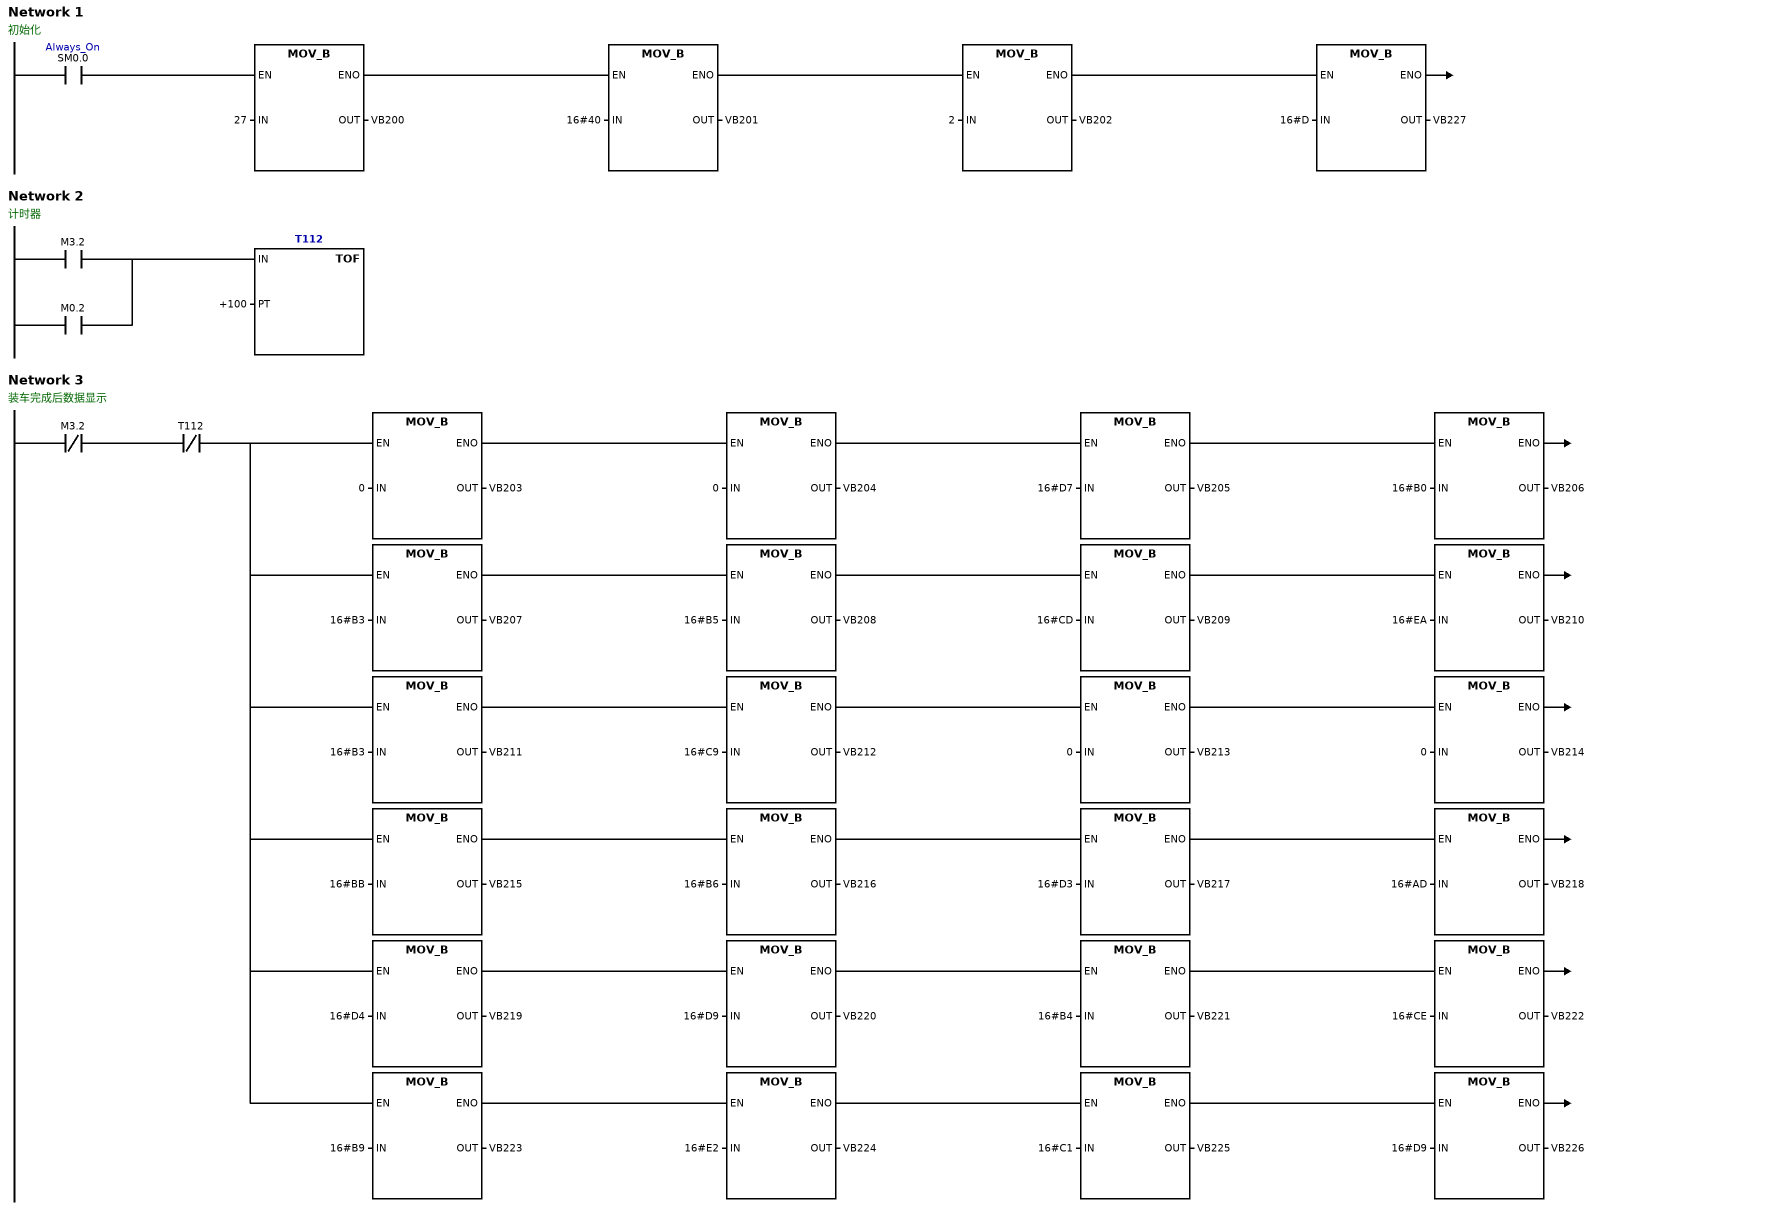
Network 1
// 初始化
LD     Always_On:SM0.0
MOVB   27, VB200
AENO
MOVB   16#40, VB201
AENO
MOVB   2, VB202
AENO
MOVB   16#D, VB227
Network 2
// 计时器
LD     M3.2
O      M0.2
TOF    T112, +100
Network 3
// 装车完成后数据显示
LDN    M3.2
AN     T112
LPS
MOVB   0, VB203
AENO
MOVB   0, VB204
AENO
MOVB   16#D7, VB205
AENO
MOVB   16#B0, VB206
LRD
MOVB   16#B3, VB207
AENO
MOVB   16#B5, VB208
AENO
MOVB   16#CD, VB209
AENO
MOVB   16#EA, VB210
LRD
MOVB   16#B3, VB211
AENO
MOVB   16#C9, VB212
AENO
MOVB   0, VB213
AENO
MOVB   0, VB214
LRD
MOVB   16#BB, VB215
AENO
MOVB   16#B6, VB216
AENO
MOVB   16#D3, VB217
AENO
MOVB   16#AD, VB218
LRD
MOVB   16#D4, VB219
AENO
MOVB   16#D9, VB220
AENO
MOVB   16#B4, VB221
AENO
MOVB   16#CE, VB222
LPP
MOVB   16#B9, VB223
AENO
MOVB   16#E2, VB224
AENO
MOVB   16#C1, VB225
AENO
MOVB   16#D9, VB226
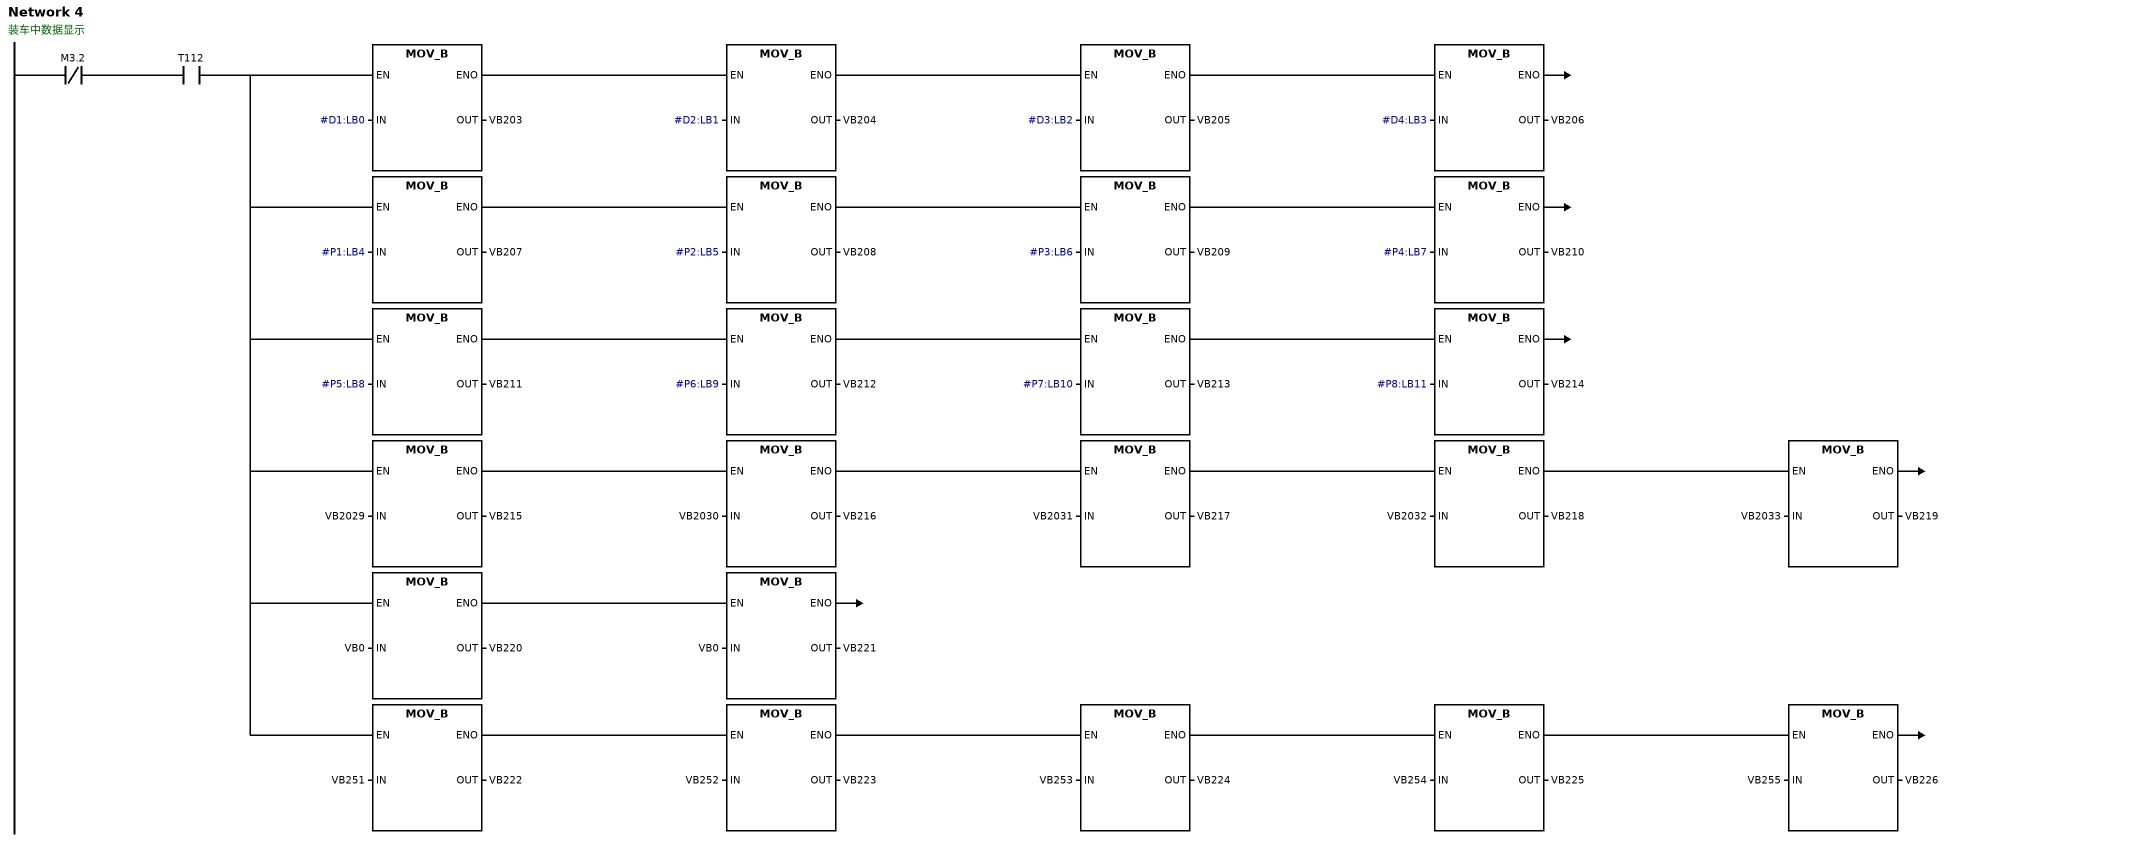
Network 4
// 装车中数据显示
LDN    M3.2
A      T112
LPS
MOVB   #D1:LB0, VB203
AENO
MOVB   #D2:LB1, VB204
AENO
MOVB   #D3:LB2, VB205
AENO
MOVB   #D4:LB3, VB206
LRD
MOVB   #P1:LB4, VB207
AENO
MOVB   #P2:LB5, VB208
AENO
MOVB   #P3:LB6, VB209
AENO
MOVB   #P4:LB7, VB210
LRD
MOVB   #P5:LB8, VB211
AENO
MOVB   #P6:LB9, VB212
AENO
MOVB   #P7:LB10, VB213
AENO
MOVB   #P8:LB11, VB214
LRD
MOVB   VB2029, VB215
AENO
MOVB   VB2030, VB216
AENO
MOVB   VB2031, VB217
AENO
MOVB   VB2032, VB218
AENO
MOVB   VB2033, VB219
LRD
MOVB   VB0, VB220
AENO
MOVB   VB0, VB221
LPP
MOVB   VB251, VB222
AENO
MOVB   VB252, VB223
AENO
MOVB   VB253, VB224
AENO
MOVB   VB254, VB225
AENO
MOVB   VB255, VB226
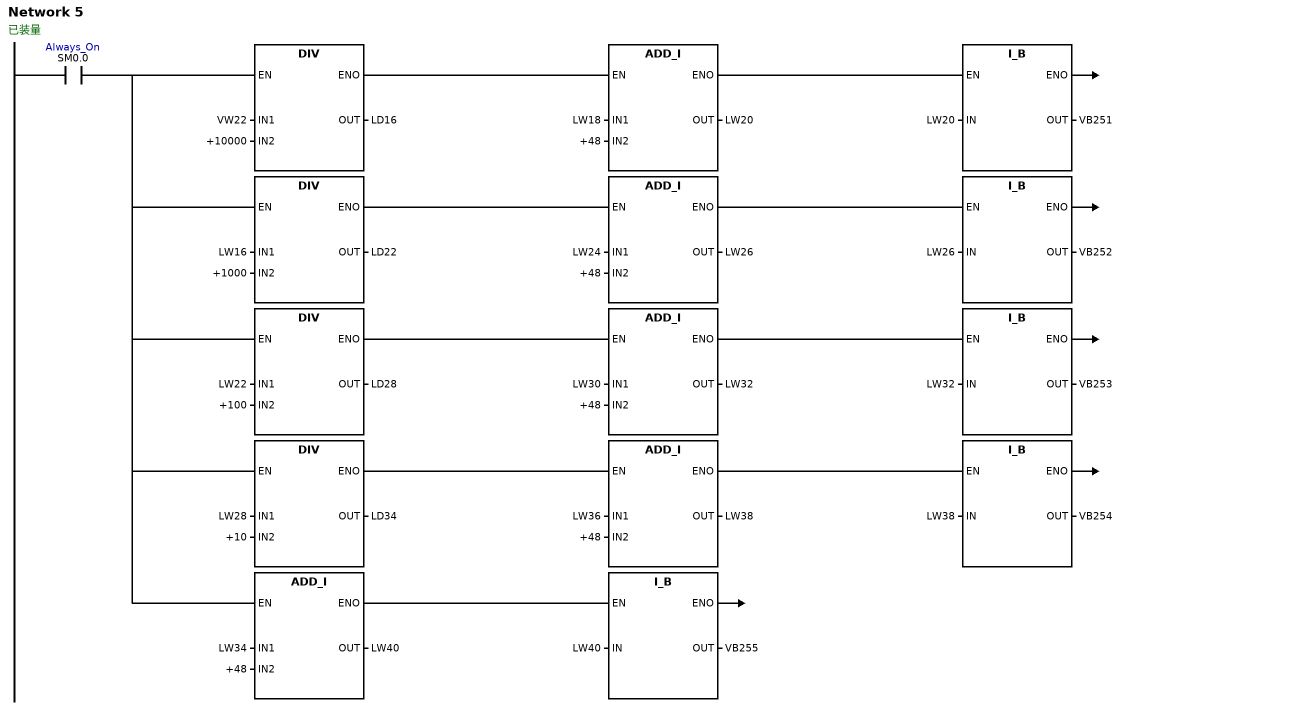
Network 5
// 已装量
LD     Always_On:SM0.0
LPS
MOVW   VW22, LW18
AENO
DIV    +10000, LD16
AENO
MOVW   LW18, LW20
AENO
+I     +48, LW20
AENO
ITB    LW20, VB251
LRD
MOVW   LW16, LW24
AENO
DIV    +1000, LD22
AENO
MOVW   LW24, LW26
AENO
+I     +48, LW26
AENO
ITB    LW26, VB252
LRD
MOVW   LW22, LW30
AENO
DIV    +100, LD28
AENO
MOVW   LW30, LW32
AENO
+I     +48, LW32
AENO
ITB    LW32, VB253
LRD
MOVW   LW28, LW36
AENO
DIV    +10, LD34
AENO
MOVW   LW36, LW38
AENO
+I     +48, LW38
AENO
ITB    LW38, VB254
LPP
MOVW   LW34, LW40
AENO
+I     +48, LW40
AENO
ITB    LW40, VB255
